TYPE "OP40_Data"
VERSION : 0.1
   STRUCT
      AssemblyResult : Byte;
      SN : String[30];
      ProcessData : "WriteProcessData";
   END_STRUCT;

END_TYPE

